{attribute 'GeneratedUsingTerminal: EL3773-0000-0016'}
{attribute addProperty BoxType "EL3773-0000-0016"}
{attribute addProperty Id "U2_SAMPLESAT %I*U2_SAMPLES_2D13B74B20"}
{attribute addProperty CRC "3641772478"}
{attribute addProperty Size "20"}
TYPE L2_Voltage_Samples_D91109BE :
STRUCT
	{attribute addProperty Name "U2_SAMPLES"}
	U2_SAMPLES AT %I* : U2_SAMPLES_2D13B74B;
END_STRUCT
END_TYPE

(* stored: Version 1.2.0.0, ProductVersion 3.1.4024.9
   DUT L2_Voltage_Samples_D91109BE: Id {2ac46f06-f52c-42d9-88ee-c85340e45738} *)
